VAR_GLOBAL
END_VAR

(* stored: Version 1.1.0.1, ProductVersion 3.1.0.19
   GVL CHD_CmdState: Id {18f471d1-5df5-4613-887e-ba1b5c405781} *)
